INTERFACE ITF_CommunicationModul

METHOD M_Connect : BOOL
VAR_INPUT
END_VAR
END_METHOD

METHOD M_Disconnect : BOOL
VAR_INPUT
END_VAR
END_METHOD

METHOD M_ResetConnection : BOOL
VAR_INPUT
END_VAR
END_METHOD

PROPERTY P_bConnected : BOOL
GET
END_GET
END_PROPERTY

END_INTERFACE

(* stored: Version 1.1.0.1, ProductVersion 3.1.4026.18
   Itf ITF_CommunicationModul: Id {4810cc8a-bb2f-4d01-ae10-324af9a1a648}
   Method M_Connect: Id {fe4f8274-1518-420a-a4d9-823324d5e171}
   Method M_Disconnect: Id {a70ffb50-a951-4357-9f6a-b5d1dce3db76}
   Method M_ResetConnection: Id {76324a3a-2abd-4da4-8e05-8b1c6dd1b8ff}
   Property P_bConnected: Id {e542eef6-d03f-474c-9b54-7da305f7da18}
   Get Get: Id {c9d93277-aa15-4ceb-952c-e7bed8bdcac4} *)
